FUNCTION_BLOCK OneSpeed_Override
VAR_INPUT
	Master_Speed : REAL;
	Pump_Ovr: BOOL;
	OA_Speed: REAL;
	OA_SpeedMin: REAL;
	OA_SpeedMax: REAL;
	
END_VAR
VAR_OUTPUT
	VSD_Speed: REAL;
	
END_VAR
VAR
END_VAR

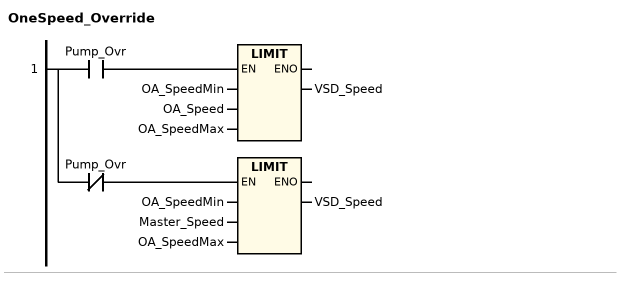
// NETWORK 1
IF Pump_Ovr THEN VSD_Speed := LIMIT(OA_SpeedMin, OA_Speed, OA_SpeedMax); END_IF
IF NOT Pump_Ovr THEN VSD_Speed := LIMIT(OA_SpeedMin, Master_Speed, OA_SpeedMax); END_IF

END_FUNCTION_BLOCK

(* stored: Version 1.1.0.1, ProductVersion 3.1.4024.12
   POU OneSpeed_Override: Id {aa335a1b-3983-4c1a-8871-f12146781783}, SpecialFunc None *)
